INTERFACE ValueWithType EXTENDS __SYSTEM.IQueryInterface

{attribute 'monitoring' := 'call'}
PROPERTY ValueType : ValueType
GET
END_GET
END_PROPERTY

END_INTERFACE

(* stored: Version 1.1.0.1, ProductVersion 3.1.4024.15
   Itf ValueWithType: Id {fc6a283b-022e-4806-bd75-e2d56e43f80a}
   Property ValueType: Id {4ee1d9d0-c89f-454b-83a2-53c3f3807e14}
   Get Get: Id {8394b104-970b-4e5a-bcf4-67612d32f55c} *)
